// TIA Portal V16 export
// export: Created 2021-11-12T13:32:46.2287407Z, ExportSetting WithDefaults, DisplayName Totally Integrated Automation Portal, DisplayVersion V16 Update 3, DisplayName TIA Portal Version Control Interface, DisplayVersion V16 Update 2, DisplayName TIA Portal Openness, DisplayVersion V16 Update 3, DisplayName SINAMICS Startdrive Advanced, DisplayVersion V16 Update 5, DisplayName SINAMICS Startdrive G130, G150, S120, S150, SINAMICS MV, S210, DisplayVersion V16 Update 5, DisplayName SINAMICS Startdrive G110M, G120, G120C, G120D, G120P, G115D, DisplayVersion V16 Update 5, DisplayName STEP 7 Professional, DisplayVersion V16 Update 3, DisplayName STEP 7 Safety, DisplayVersion V16, DisplayName WinCC UA Professional, DisplayVersion V16 Update 3
DATA_BLOCK "HMI_PARAM_Zone200"   // DB24
{ S7_Optimized_Access := 'TRUE'; DB_Accessible_From_OPC_UA := 'FALSE' }
VERSION : 0.1
// stored: AutoNumber true, DBAccessibleFromOPCUA false, IsOnlyStoredInLoadMemory false, IsRetainMemResEnabled false, IsWriteProtectedInAS false, MemoryReserve 100
   VAR
      Mode : "UDT_Zone_Parameter";   // Parameters of zone 200
      Station210_Mode : "UDT_Station_Parameter";   // Parameters of station 210
      Station220_Mode : "UDT_Station_Parameter";   // Parameters of station 220
      Station230_Mode : "UDT_Station_Parameter";   // Parameters of station 230
      Station2R1_Mode : "UDT_Station_Parameter";   // Parameters of station 2R1
      Station2R2_Mode : "UDT_Station_Parameter";   // Parameters of station 2R2
      StationSCH1_Mode : "UDT_Station_Parameter";   // Parameters of forging station SCH1
      StationBSN3_Mode { S7_SetPoint := 'True'} : "UDT_Station_Parameter";   // Parameters of furnace station BSN1
      xxxxx___Alarms___xxxxx { S7_SetPoint := 'True'} : Byte;
      "200UF01-SF01" : "UDT_DI_Mon_Parameter";   // E-stop 200UF01-SF01
      "200QQ01_ES" { S7_SetPoint := 'True'} : "UDT_DI_Mon_Parameter";   // E-stop gate 200QQ01
      "200QQ02_ES" { S7_SetPoint := 'True'} : "UDT_DI_Mon_Parameter";   // E-stop gate 200QQ02
      "200QQ03_ES" { S7_SetPoint := 'True'} : "UDT_DI_Mon_Parameter";   // E-stop gate 200QQ03
      "200QQ04_ES" { S7_SetPoint := 'True'} : "UDT_DI_Mon_Parameter";   // E-stop gate 200QQ04
      "200QQ05_ES" { S7_SetPoint := 'True'} : "UDT_DI_Mon_Parameter";   // E-stop gate 200QQ05
      "200RU01-KF01" { S7_SetPoint := 'True'} : "UDT_DI_Mon_Parameter";   // gate module 200RU01-KF01
      "200RU01-KF02" { S7_SetPoint := 'True'} : "UDT_DI_Mon_Parameter";   // gate module 200RU01-KF02
      "200RU01-KF03" { S7_SetPoint := 'True'} : "UDT_DI_Mon_Parameter";   // gate module 200RU01-KF03
      "200RU01-KF04" { S7_SetPoint := 'True'} : "UDT_DI_Mon_Parameter";   // gate module 200RU01-KF04
   END_VAR
BEGIN
   Mode.HMI1.FuncBtnPanelNr := 10;
   Mode.HMI2.FuncBtnPanelNr := 20;
   Mode.HMI3.FuncBtnPanelNr := 30;
END_DATA_BLOCK
